// Mitsubishi GX Works2 project: CydeusPlatform2   PLC: FX3U/FX3UC

TYPE ST_1SolCylinderInterface : STRUCT
  bBusy : BOOL;
  bError : BOOL;
  bDone : BOOL;
  bGoActive : BOOL;
  bReset : BOOL;
  tDelayTime : TIME;
  tTimeout : TIME;
END_STRUCT END_TYPE

TYPE ST_ServoMotorInterface : STRUCT
  bBusy : BOOL;
  bError : BOOL;
  bDone : BOOL;
  bServoEnabled : BOOL;
  bEnable : BOOL;
  bStop : BOOL;
  bAbort : BOOL;
  bReset : BOOL;
  bJogPos : BOOL;
  bJogNeg : BOOL;
  bMoveRel : BOOL;
  rMoveDist : REAL;
  iMoveVel : DINT;
  iMoveAccel : DINT;
END_STRUCT END_TYPE

// global labels: GVL_Error
VAR_GLOBAL
  arrError : ARRAY [0..9] OF BOOL;
END_VAR
VAR_GLOBAL CONSTANT
  uiNumErrMinus1 : INT := 9;
END_VAR

// global labels: GVL_Main
VAR_GLOBAL
  bAlarmTrigger : BOOL;
  bMachineError : BOOL;
  bManualMode : BOOL;
  bAutoMode : BOOL;
  bStepMode : BOOL;
  bSimMode : BOOL;
  objPunching : CL_1Sol1SenCylinder;
  stServoMotor : ST_ServoMotorInterface;
  stPunching : ST_1SolCylinderInterface;
  objServoMotor : CL_ServoMotor;
END_VAR

// global labels: GVL_HMI
VAR_GLOBAL
  btnPunchingOutput : BOOL;
  btnPowerMotor : BOOL;
  btnManualMode : BOOL;
  btnInitialize : BOOL;
  btnAutoMode : BOOL;
  btnAbort : BOOL;
  btnStepMode : BOOL;
  btnBack : BOOL;
  btnTest : BOOL;
  btnTestManualOn : BOOL;
  btnSetup : BOOL;
  btnReset : BOOL;
  btnStartAuto : BOOL;
  tboxPulsePerRev AT D200 : DINT;
  tboxRadius AT D202 : REAL;
  tboxMoveVel AT D204 : DINT;
  tboxMoveAccel AT D206 : DINT;
  tboxPunchingDelayTime AT D210 : TIME;
  tboxPunchingTimeout AT D212 : TIME;
  btnServoStop : BOOL;
  btnServoEnable : BOOL;
  btnServoAbort : BOOL;
  btnServoReset : BOOL;
  btnServoJogPos : BOOL;
  btnServoJogNeg : BOOL;
  btnServoMoveRel : BOOL;
  tboxMoveDist : REAL;
END_VAR

// global labels: GVL_Output
VAR_GLOBAL
  boPunchingOutput AT Y006 : BOOL;
  boPowerMotor AT Y007 : BOOL;
  bMaPunchingOutput : BOOL;
  bMaPowerMotor : BOOL;
  bAuPunchingOutput : BOOL;
  bAuPowerMotor : BOOL;
  boServoPP AT Y000 : BOOL;
  boServoNP AT Y001 : BOOL;
  boServoSON AT Y004 : BOOL;
  boServoRES AT Y005 : BOOL;
  boServoEM2 AT Y003 : BOOL;
END_VAR

// global labels: GVL_Input
VAR_GLOBAL
  biEstop1 AT X000 : BOOL;
  biEstop2 AT X001 : BOOL;
  biPunchingTriggered AT X002 : BOOL;
  biFeederSensor AT X003 : BOOL;
  biServoINP AT X005 : BOOL;
  biServoRD AT X006 : BOOL;
  biServoALM AT X007 : BOOL;
  bEstop1 : BOOL;
  bEstop2 : BOOL;
  bPunchingTriggered : BOOL;
  bFeederSensor : BOOL;
  bServoINP : BOOL;
  bServoRD : BOOL;
  bServoALM : BOOL;
  biPunchingDone AT X004 : BOOL;
  bPunchingDone : BOOL;
END_VAR

// global labels: GVL_System
VAR_GLOBAL
  bCommandComplete AT M8029 : BOOL;
END_VAR

// task Task_01 (event TRUE, interval 0, priority 31): MAIN

PROGRAM MAIN
VAR
  fbErrorController : FB_ErrorController;
  fbOutputController : FB_OutputController;
  fbManualMode : FB_ManualMode;
  fbStateMachine : FB_StateMachine;
  fbInputLinker : FB_InputLinker;
  fbObjectExecution : FB_ObjectExecution;
END_VAR
(*Input Linker*)
fbInputLinker();

(*State Machine*)
fbStateMachine();

(*Object Execution*)
fbObjectExecution();

(*Output Controller*)
fbOutputController();

(*Error Controller*)
fbErrorController(bResetError := btnReset);
bMachineError := fbErrorController.bError;
END_PROGRAM

FUNCTION_BLOCK FB_ErrorController
VAR
  ii : INT;
END_VAR
VAR_OUTPUT
  bError : BOOL;
END_VAR
VAR_INPUT
  bResetError : BOOL;
END_VAR
(*Error Controller*)

(*Reset Errors*)
IF bResetError THEN
	FOR ii := 0 TO uiNumErrMinus1  DO
		arrError[ii] := FALSE;
	END_FOR;
END_IF;

(*Register Errors*)
SET(bAlarmTrigger, arrError[0]);

(*Machine Error Trigger*)
bError := FALSE;
FOR ii := 0 TO uiNumErrMinus1  DO
	bError := bError OR arrError[ii];
END_FOR;
END_FUNCTION_BLOCK

FUNCTION FUN_Output
VAR_INPUT
  b_OutAuto : BOOL;
  b_OutMan : BOOL;
  b_ManualMode : BOOL;
END_VAR
FUN_Output := (b_ManualMode AND b_OutMan) OR (NOT b_ManualMode AND b_OutAuto);
END_FUNCTION

FUNCTION_BLOCK FB_OutputController
(*Output Controller*)

(*Calculate the logical output, then assign to physical output*)
boPowerMotor := FUN_Output(bManualMode, bAuPowerMotor, bMaPowerMotor);
boPunchingOutput := FUN_Output(bManualMode, bAuPunchingOutput, bMaPunchingOutput);
END_FUNCTION_BLOCK

FUNCTION_BLOCK FB_ManualMode
VAR_INPUT
  bEnable : BOOL;
END_VAR
(*Manual Mode*)

(*Enable Manual Mode*)
bManualMode := btnManualMode;

(*Hold Current status of Outputs*)
;;;;;;

(*Buttons on HMI control logical outputs*)
IF bManualMode THEN
	bMaPowerMotor := btnPowerMotor;
	bMaPunchingOutput := btnPunchingOutput;
END_IF;

(*Buttons on HMI control servo motor*)
IF bManualMode THEN
	stServoMotor.bAbort := btnServoAbort;
	stServoMotor.bEnable := btnServoEnable;
	stServoMotor.bStop := btnServoStop;
	stServoMotor.bReset := btnServoReset;
	stServoMotor.bJogPos := btnServoJogPos;
	stServoMotor.bJogNeg := btnServoJogNeg;
	stServoMotor.bMoveRel := btnServoMoveRel;
	stServoMotor.rMoveDist := tboxMoveDist;
END_IF;
END_FUNCTION_BLOCK

FUNCTION_BLOCK FB_Initializing
VAR_OUTPUT
  bDone : BOOL;
END_VAR
VAR_INPUT
  bEnable : BOOL;
END_VAR
VAR
  iState : DINT;
END_VAR
VAR_OUTPUT
  bAbort : BOOL;
END_VAR
VAR
  fbDelayStep0 : TON;
  fbDelayStep10 : TON;
  bResetFB : BOOL;
END_VAR
(*Initializing*)
PLS(bEnable, bResetFB);
IF bResetFB THEN
	iState := 0;
END_IF;

IF bEnable THEN
		CASE iState OF
				0: 	(*Home the punching*)
						IF stPunching.bDone OR fbDelayStep0.Q THEN
								iState := 10;
						END_IF;
						
				10:	(*Servo ON*)
						IF stServoMotor.bServoEnabled THEN
								iState := 20;
						ELSIF fbDelayStep10.Q THEN
								iState := 50;
						END_IF;
						
				20: 	(*Done*)
						;
				50: 	(*Abort*)	
						;
		END_CASE;
		
		RST((iState = 0), stPunching.bGoActive);
		SET((iState = 10), stServoMotor.bEnable);
END_IF;

bDone := iState = 20 AND bEnable;
bAbort := iState = 50 AND bEnable;				

fbDelayStep0(IN := iState = 0 AND bEnable, PT := t#2s);
fbDelayStep10(IN := iState = 10 AND bEnable, PT := t#5s);
END_FUNCTION_BLOCK

FUNCTION_BLOCK FB_StateMachine
VAR
  iState : INT;
  fbInitializing : FB_Initializing;
  fbAutoMode : FB_AutoMode;
  fbManualMode : FB_ManualMode;
  iLastState : INT;
  bInitializingDone : BOOL;
  bAutoModeReturn : BOOL;
  bManualModeReturn : BOOL;
  bInitializingAbort : BOOL;
END_VAR
(*Main State Machine*)
IF (btnAbort OR bMachineError) AND NOT (iState = 1) AND NOT (iState >= 10) THEN	(*Abort command*)
	iState := 0;
END_IF;

CASE iState OF
	0: 		(*Aborting*)
		iState := 1;
	
	1: 		(*Begin*)
		IF btnInitialize AND NOT bMachineError THEN
			iState := 2;
		ELSIF btnTest THEN
			iLastState := iState;
			iState := 10;
		ELSIF btnSetup THEN
			iLastState := iState;
			iState := 15;
		END_IF;
		
	2: 		(*Initializing*)
		IF bInitializingDone AND NOT bMachineError THEN
			iState := 3;
		ELSIF bInitializingAbort THEN
			iState := 0;
		END_IF;
		
	3: 		(*Ready*)
		IF btnAutoMode AND NOT bMachineError THEN
			iState := 4;
		ELSIF btnStepMode AND NOT bMachineError THEN
			iState := 5;
		ELSIF btnManualMode AND NOT bMachineError THEN
			iState := 6;
		ELSIF btnTest THEN
			iLastState := iState;
			iState := 10;
		END_IF;
	
	4: 		(*Running Auto Mode*)
		IF bAutoModeReturn  AND NOT bMachineError THEN
			iState := 3;
		END_IF;
		
	5: 		(*Running Step Mode*)
		IF bAutoModeReturn AND NOT bMachineError THEN
			iState := 3;
		END_IF;
		
	6: 		(*Running Manual Mode*)
		IF btnBack AND NOT bMachineError THEN
			iState := 3;
		END_IF;
		
	10: 		(*Testing*)
		IF btnBack THEN
			iState := iLastState;
		END_IF;
		
	15: 		(*Setting*)
		IF btnBack THEN
			iState := iLastState;
		END_IF;
	
ELSE 
		;
END_CASE;

(*State Action*)
bAutoMode := iState = 4;
bStepMode := iState = 5;
bManualMode := iState = 6;

(*Function Block Call*)
fbInitializing(bEnable := iState = 2,
						bDone := bInitializingDone,
						bAbort := bInitializingAbort);
fbAutoMode(bEnable := (iState = 4) OR (iState = 5),	
							bEnStepMode := iState = 5,
							bReset := iState = 0,
							bReturn := bAutoModeReturn);
fbManualMode(bEnable := (iState = 6) OR (iState = 10 AND btnTestManualOn));
END_FUNCTION_BLOCK

FUNCTION_BLOCK FB_AutoMode
VAR_OUTPUT
  bReturn : BOOL;
END_VAR
VAR_INPUT
  bEnStepMode : BOOL;
  bEnable : BOOL;
  bReset : BOOL;
END_VAR
VAR
  bResetFB : BOOL;
  iState : INT;
  bState80 : BOOL;
END_VAR
VAR_INPUT
  bNext : BOOL;
END_VAR
VAR
  bNextStep : BOOL;
END_VAR
(*Initialize and Reset Function Block*)
PLS((bReset OR bEnable), bResetFB);
IF bResetFB THEN
	iState := 0;
END_IF;

(*Auto Mode State Machine*)
CASE iState OF
		0: 		(*Ready*)
				IF btnStartAuto THEN
					iState := 10;
				END_IF;
				
		10: 		(*Wait for raw material*)
				IF bFeederSensor AND bNextStep THEN
					iState := 20;
				END_IF;
				
		20: 		(*Cut spare material before beginning*)
				IF bPunchingTriggered  THEN
					iState := 30;
				END_IF;
				
		30: 		(*Wait for Punching done*)
				IF stPunching.bDone AND bNextStep THEN
					iState := 40;
				END_IF;
		
		40: 		(*Feed new raw material to punching machine*)
				IF stServoMotor.bDone AND bNextStep THEN
					iState := 50;
				END_IF;
			
		50: 		(*Cut raw material into final product*)
				IF bPunchingTriggered THEN
					iState := 60;
				END_IF;
				
		60: 		(*Wait for Punching done*)
				IF stPunching.bDone AND bNextStep THEN
					iState := 70;
				END_IF;

		70: 		(*Check for raw material*)
				IF bFeederSensor THEN
					iState := 40;
				ELSE 
					iState := 80;
				END_IF;
				
		80: 		(*FB Return*)
				PLS(TRUE, bState80);
				IF NOT bState80 THEN
					iState := 0;
				END_IF;
				
END_CASE;

(*Auto Mode State Action*)
bReturn := iState = 80 AND bEnable;
bNextStep := (NOT bEnStepMode OR (bEnStepMode AND bNext)) AND bEnable;

stServoMotor.bMoveRel := (iState = 40);
stPunching.bGoActive := (iState = 20) OR (iState = 30) OR (iState = 50) OR (iState = 60);
END_FUNCTION_BLOCK

FUNCTION_BLOCK FB_InputLinker
(*Input Linker*)

(*Link physical input to logical input memory*)
IF NOT bSimMode THEN	
		bEstop1 := biEstop1;
		bEstop2 := biEstop2;
		bPunchingTriggered := biPunchingTriggered;
		bFeederSensor := biFeederSensor;
		bPunchingDone := biPunchingDone;
		bServoINP := biServoINP;
		bServoRD := biServoRD;
		bServoALM := biServoALM;
END_IF;
END_FUNCTION_BLOCK

FUNCTION_BLOCK FB_ObjectExecution
objServoMotor(biINP := bServoINP,
								biRD := bServoRD,
								biALM := bServoALM,
								boNPz := boServoNP,
								boEM2 := boServoEM2,
								boRES := boServoRES,
								boSON := boServoSON,
								
								bEnable := stServoMotor.bEnable,
								bStop := stServoMotor.bStop,
								bAbort := stServoMotor.bAbort,
								bReset := stServoMotor.bReset,
								iOutChannel := 0,
								iMoveDelay := 100,
								iPulsePerRev := tboxPulsePerRev,
								rRadius := tboxRadius,
								
								bJogPos := stServoMotor.bJogPos,
								bJogNeg := stServoMotor.bJogNeg,
								
								bMoveRel := stServoMotor.bMoveRel,
								rMoveDist := stServoMotor.rMoveDist,
								iMoveVel := tboxMoveVel,
								iMoveAccel := tboxMoveAccel,

								bBusy := stServoMotor.bBusy,
								bDone := stServoMotor.bDone,
								bError := stServoMotor.bError,
								bServoEnabled := stServoMotor.bServoEnabled);
								
								
objPunching(biSensorDone := bPunchingDone,
							biActiveFeedback := bPunchingTriggered,
							boSolenoid := bMaPunchingOutput,
							
							bGoActive := stPunching.bGoActive,
							bReset := stPunching.bReset,
							tDelayTime := tboxPunchingDelayTime,
							tTimeout := tboxPunchingTimeout,

							bBusy := stPunching.bBusy,
							bInHomePos := stPunching.bDone,
							bError := stPunching.bError);
END_FUNCTION_BLOCK

FUNCTION_BLOCK CL_1Sol1SenCylinder
VAR_INPUT
  biSensorDone : BOOL;
  bGoActive : BOOL;
  bReset : BOOL;
END_VAR
VAR_OUTPUT
  boSolenoid : BOOL;
  bBusy : BOOL;
  bInHomePos : BOOL;
  bError : BOOL;
END_VAR
VAR_INPUT
  tDelayTime : TIME;
  tTimeout : TIME;
END_VAR
VAR
  fbDelayTime : TON;
  fbTimeout : TON;
END_VAR
VAR_INPUT
  biActiveFeedback : BOOL;
END_VAR
VAR
  bSensorDoneHold : BOOL;
  bBusyPulse : BOOL;
END_VAR
(*Activate Output: Enable solenoid on valve*) 
boSolenoid := bGoActive;

(*Process Input: Wait for sensors signal*)
PLS(bBusy, bBusyPulse);
SET(biSensorDone, bSensorDoneHold);
RST(bBusyPulse, bSensorDoneHold);
bInHomePos := fbDelayTime.Q AND NOT bSensorDoneHold;
bBusy := biActiveFeedback AND NOT biSensorDone;

(*Error handling*)
		(*Notify timeout error*)
		SET(fbTimeout.Q, bError);

		(*Reset timeout error*)
		RST(bReset, bError);

(*Timers call*)
fbDelayTime(IN := NOT bBusy, PT := tDelayTime);
fbTimeout(IN := bBusy, PT := tTimeout);
END_FUNCTION_BLOCK

FUNCTION_BLOCK CL_ServoMotor
VAR_INPUT
  biINP : BOOL;
  biRD : BOOL;
  biALM : BOOL;
  bEnable : BOOL;
  bStop : BOOL;
  bAbort : BOOL;
  bReset : BOOL;
  bJogPos : BOOL;
  bJogNeg : BOOL;
  bMoveRel : BOOL;
  rMoveDist : REAL;
END_VAR
VAR_OUTPUT
  boNPz : BOOL;
  boEM2 : BOOL;
  boSON : BOOL;
  boRES : BOOL;
  bBusy : BOOL;
  bError : BOOL;
  bDone : BOOL;
  bServoEnabled : BOOL;
END_VAR
VAR
  iState : INT;
  fbResetHold : TP_10;
  bResetHold : BOOL;
  fbMoveDelay : TON;
END_VAR
VAR_INPUT
  iMoveDelay : WORD;
END_VAR
VAR
  tMoveDelay : TIME;
  iStopState : INT;
END_VAR
VAR_INPUT
  iMoveVel : DINT;
  iMoveAccel : DINT;
  iPulsePerRev : DINT;
  rRadius : REAL;
END_VAR
VAR
  iFrequency : DINT;
  iPulse : DINT;
  iAccel : DINT;
  bOutPulse : BOOL;
END_VAR
VAR_INPUT
  iOutChannel : INT;
END_VAR
(*Procedure*)
		(*Abort*)
		IF bAbort OR NOT bEnable OR bError THEN
				iState := 0;
				iStopState := 0;
		END_IF;
		
		(*Reset*)
		IF bReset AND bError THEN
				iState := 0;
				iStopState := 0;
		END_IF;		
		
		(*Stop*)
		CASE iStopState OF
				0: 	(*Wait for stop signal*)
						IF bStop THEN
								iStopState := 10;
						END_IF;
						
				10: 	(*Execute Stop*)
						IF iState > 20 THEN
								iState := 20;
						END_IF;
						IF biINP THEN
								iStopState := 20;
						END_IF;
						
				20: 	(*Stop done, wait for command release*)
						IF NOT bStop THEN
								iStopState := 0;
						END_IF;
		END_CASE;	
						

(*Main State Machine*)
CASE iState OF 
		0: 	(*Unenabled, wait for Enable command*)
				IF bEnable AND NOT bStop AND NOT bError THEN
						iState := 10;
				END_IF;
				
		10: 	(*Servo On*)
				IF bServoEnabled THEN
						iState := 20;
				END_IF;
						
		20: 	(*Servo Ready, wait for moving command*)
				IF bJogPos AND NOT bStop AND NOT bError THEN
						iState := 100;
				ELSIF bJogNeg AND NOT bStop AND NOT bError THEN
						iState := 150;
				ELSIF bMoveRel AND NOT bStop AND NOT bError THEN
						iState := 200;
				END_IF;
				
		100: 	(*Calculate number of pulse*)			
				iFrequency := iPulsePerRev;
				iPulse := 0;	
				iAccel := iMoveAccel;
				iState := 110;
				
		110: 	(*Execute Jog Pos command*)
				IF NOT bJogPos THEN 
						iState := 20;
				END_IF;
				
		150: 	(*Execute Jog Neg command*)
				IF NOT bJogNeg THEN
						iState := 20;
				END_IF;
				
		200: 	(*Calculate number of pulse*)
				iFrequency := REAL_TO_DINT(DINT_TO_REAL(iPulsePerRev*iMoveVel)/60.0);
				iPulse := REAL_TO_DINT(DINT_TO_REAL(iPulsePerRev)*rMoveDist/(2.0*3.1415926*rRadius));	
				iAccel := iMoveAccel;
				tMoveDelay := WORD_TO_TIME(iMoveDelay);
				iState := 210;
		
		210: 	(*Execute Move Relative command*)
				IF biINP AND fbMoveDelay.Q THEN
						iState := 220;
				END_IF;		
				
		220: 	(*Move Relative done, wait for command release*)
				IF NOT bMoveRel THEN
						iState := 20;
				END_IF;
				
END_CASE;
	
(*State Action*)
		boSON := (bEnable AND iState >= 10 AND NOT bAbort);			(*Enable Servo Motor*)	
		boEM2 := NOT bAbort OR NOT biALM;											(*Abort Servo Motor*)
		boRES := fbResetHold.Q AND NOT biALM;									(*Reset Servo Motor*)		
		
		bBusy := (iState = 110) OR (iState = 150) OR (iState = 210) OR (iStopState = 10);
		bDone := (iState = 220) OR (iStopState = 20);									(*Servo movement is done*)
		bServoEnabled := biRD;																		(*Servo is powered on*)
	
		SET(NOT biALM, bError);																		(*Notify Servo Motor Error*)
		RST((bReset AND bError), bError);													(*Reset object error*)	
		
		bOutPulse := ((iState = 110) OR (iState = 150) OR (iState = 210)) AND NOT (iStopState = 10);	(*Enable Pulse*)
		boNPz := ((iState = 150) OR (rMoveDist < 0.0));
	
(*Function Block Call*)
bResetHold := (bReset AND NOT fbResetHold.Q) OR (bResetHold AND fbResetHold.Q) ;
fbResetHold(IN := bResetHold, PT := t#600ms);
fbMoveDelay(IN := bMoveRel AND bServoEnabled AND NOT bStop AND NOT bAbort AND NOT bError, PT := tMoveDelay);

CASE iOutChannel OF 
		0: 	(*Y000*)
				DPLSR(bOutPulse, iFrequency, iPulse, iAccel, Y000);
		1:		(*Y001*)
				DPLSR(bOutPulse, iFrequency, iPulse, iAccel, Y001);
		2:		(*Y002*)
				DPLSR(bOutPulse, iFrequency, iPulse, iAccel, Y002);
END_CASE;
END_FUNCTION_BLOCK

FUNCTION_BLOCK FB_Aborting
VAR
  bEnable : BOOL;
  bDone : BOOL;
END_VAR
(*Aborting*)
IF bEnable THEN
		;
END_IF;
END_FUNCTION_BLOCK
